FUNCTION_BLOCK FB_Assigner
VAR_INPUT
	i_TagAssignment : I_TagAssignment;
END_VAR
VAR_OUTPUT
END_VAR
VAR
END_VAR

IF i_TagAssignment <> 0 THEN
		THIS^.i_TagAssignment := i_TagAssignment;
END_IF	
	


i_TagAssignment.R1();
i_TagAssignment.R2();
i_TagAssignment.R3();
i_TagAssignment.R4();
i_TagAssignment.R5();
i_TagAssignment.AA1();
i_TagAssignment.AA2();
i_TagAssignment.DCM();
i_TagAssignment.MVA();
i_TagAssignment.MVB();
i_TagAssignment.RV();

END_FUNCTION_BLOCK

(* stored: Version 1.1.0.1, ProductVersion 3.1.4024.6
   POU FB_Assigner: Id {f811e592-2cf9-45e4-9aaa-764034fb0f89}, SpecialFunc None *)
